TYPE LaserVar :
STRUCT
    sv_bPLCHandShaking : BOOL;
    sv_bIPCHandShaking    : BOOL;
END_STRUCT
END_TYPE

(* stored: Version 1.1.0.1, ProductVersion 3.1.4024.15
   DUT LaserVar: Id {8c9e7e94-9a3c-42b3-bca6-728a865f69d6} *)
